TYPE "UDT_HMI_Alarm_V2"
VERSION : 0.1
   STRUCT
      t : Struct
         x0 : Bool;
         x1 : Bool;
         x2 : Bool;
         x3 : Bool;
         x4 : Bool;
         x5 : Bool;
         x6 : Bool;
         x7 : Bool;
         x8 : Bool;
         x9 : Bool;
         x10 : Bool;
         x11 : Bool;
         x12 : Bool;
         x13 : Bool;
         x14 : Bool;
         x15 : Bool;
      END_STRUCT;
      iHmiSumAlm : Word;
   END_STRUCT;

END_TYPE

DATA_BLOCK "SpeedUP_Hmi"
{ S7_Optimized_Access := 'FALSE' }
VERSION : 0.1
NON_RETAIN
   STRUCT
      tHMR { ExternalWritable := 'False'} : Struct   // {[Unit]|[Scada Unit]|[LowLimit]|[HigLimit]|[Acces]}
         xControlSnapEnabled { ExternalWritable := 'False'} : Bool;   // Control Snap Enabled {x|x|x|x|O}
         xControlSnap1 { ExternalWritable := 'False'} : Bool;   // Control Snap Photocel 1 {x|x|x|x|O}
         xControlSnap2 { ExternalWritable := 'False'} : Bool;   // Control Snap Photocel 2 {x|x|x|x|O}
         iControlSnap1 { ExternalWritable := 'False'} : Int;   // State Snap Photocel 1 (1=No anomaly, 7=Anomaly) {x|x|x|x|O}
         iControlSnap2 { ExternalWritable := 'False'} : Int;   // State Snap Photocel 2 (1=No anomaly, 7=Anomaly) {x|x|x|x|O}
      END_STRUCT;
      tHMW : Struct   // {[Unit]|[Scada Unit]|[LowLimit]|[HigLimit]|[Acces]}
         xEnableDisableControlSnap : Bool;   // Enabled/Disable control Snap {x|x|x|x|O}
      END_STRUCT;
   END_STRUCT;


BEGIN

END_DATA_BLOCK

DATA_BLOCK "SpeedUP_Alm"
{ S7_Optimized_Access := 'FALSE' }
VERSION : 0.1
   STRUCT
      tEmergencyAlarm { ExternalWritable := 'False'} : Array["STARTARRAY".."DALARM"] of "UDT_HMI_Alarm_V2";
      tAlarm { ExternalWritable := 'False'} : Array["STARTARRAY".."DALARM"] of "UDT_HMI_Alarm_V2";
      tWarning { ExternalWritable := 'False'} : Array["STARTARRAY".."DALARM"] of "UDT_HMI_Alarm_V2";
   END_STRUCT;


BEGIN

END_DATA_BLOCK

